// Hola Mundo de la Programación de PLC
PROGRAM MAIN
VAR
    ContadorCiclos: UINT;
    i_Pulsador AT %I* : BOOL;
    o_Lampara  AT %Q* : BOOL;
END_VAR

ContadorCiclos := ContadorCiclos + 1;
o_Lampara := i_Pulsador;

END_PROGRAM

(* stored: Version 1.1.0.1, ProductVersion 3.1.4024.16
   POU MAIN: Id {19ef5ada-303e-4586-a55e-29658a9ad5ab}, SpecialFunc None *)
